FUNCTION_BLOCK SS4_Laser (* Basic FB with empty ECC *)
  (* Standard: 61499-2 *)
  (* Version 1.0, 2025-08-24, DEVIASH *)
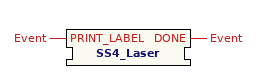
  EVENT_INPUT
    PRINT_LABEL;
  END_EVENT
  EVENT_OUTPUT
    DONE;
  END_EVENT
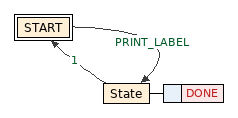
  EC_STATES
    START; (* Initial State *)
    State : -> DONE;
  END_STATES
  EC_TRANSITIONS
    START TO State := PRINT_LABEL;
    State TO START := 1;
  END_TRANSITIONS
END_FUNCTION_BLOCK
